{attribute 'qualified_only'}
{attribute 'strict'}
TYPE E_JogType :
(
	Joint,
  Cartesian
);
END_TYPE

(* stored: Version 1.1.0.1
   DUT E_JogType: Id {eb8c54f1-2aa1-4e03-814f-79d0527e577b} *)
